FUNCTION_BLOCK OR_16 (* FB to calculate bitwise boolean OR (generic FB) *)
  (* Standard: 61131-3; Classification: standard bitwise boolean function; Description: Copyright (c) 2014, 2024 Profactor GmbH, HR Agrartechnik GmbH This program and the accompanying materials are made available under the terms of the Eclipse Public License 2.0 which is available at https://www.eclipse.org/legal/epl-2.0/ SPDX-License-Identifier: EPL-2.0 *)
  (* Version 1.0, 2024-07-15, Franz Höpfinger, HR Agrartechnik GmbH, copy from OR_10 and make a OR_16 in the same way *)
  {SET_ATTRIBUTE(GenericClassName, 'GEN_OR')}
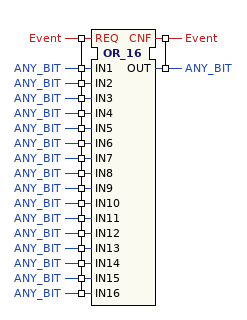
  EVENT_INPUT
    REQ WITH IN1, IN2, IN3, IN4, IN5, IN6, IN7, IN8, IN9, IN10, IN11, IN12, IN13, IN14, IN15, IN16; (* Normal Execution Request *)
  END_EVENT
  EVENT_OUTPUT
    CNF WITH OUT; (* Execution Confirmation *)
  END_EVENT
  VAR_INPUT
    IN1 : ANY_BIT; (* OR input 1 *)
    IN2 : ANY_BIT; (* OR input 2 *)
    IN3 : ANY_BIT; (* OR input 3 *)
    IN4 : ANY_BIT; (* OR input 4 *)
    IN5 : ANY_BIT; (* OR input 5 *)
    IN6 : ANY_BIT; (* OR input 6 *)
    IN7 : ANY_BIT; (* OR input 7 *)
    IN8 : ANY_BIT; (* OR input 8 *)
    IN9 : ANY_BIT; (* OR input 9 *)
    IN10 : ANY_BIT; (* OR input 10 *)
    IN11 : ANY_BIT; (* OR input 11 *)
    IN12 : ANY_BIT; (* OR input 12 *)
    IN13 : ANY_BIT; (* OR input 13 *)
    IN14 : ANY_BIT; (* OR input 14 *)
    IN15 : ANY_BIT; (* OR input 15 *)
    IN16 : ANY_BIT; (* OR input 16 *)
  END_VAR
  VAR_OUTPUT
    OUT : ANY_BIT; (* OR result *)
  END_VAR
END_FUNCTION_BLOCK
